// TwinCAT 3 PLC project Plc
// ProgramVersion: 3.1.4024.0
// libraries:
//   Tc2_Standard, * (Beckhoff Automation GmbH)
//   Tc2_System, * (Beckhoff Automation GmbH)
//   Tc3_Module, * (Beckhoff Automation GmbH)
//   VisuSymbols,3.5.10.0,System
// project tree:
//   DUTs/ E_States.TcDUT
//   / Gestore di visualizzazione.TcVMO (not stored), GlobalTextList.TcGTLO, PlcTask.TcTTO
//   GVLs/ Gvl.TcGVL
//   POUs/ FB_StateMachine.TcPOU, MAIN.TcPOU
//   VISUs/ Visualization.TcVIS
// real-time tasks:
//   TASK PlcTask: cycle T#10ms, priority 20, ADS port 350

CONFIGURATION Plc
    RESOURCE PLC ON TwinCAT3
        TASK PlcTask(INTERVAL := T#10ms, PRIORITY := 20);
        PROGRAM MAIN WITH PlcTask : MAIN;
    END_RESOURCE
END_CONFIGURATION

// ---- DUTs/E_States.TcDUT
{attribute 'qualified_only'}
{attribute 'strict'}
TYPE E_States :
(
	eStop := 0,
	eGreen,
	eYellow,
	eRed
);
END_TYPE

// ---- GVLs/Gvl.TcGVL
{attribute 'qualified_only'}
VAR_GLOBAL
	bStart: BOOL; //Pulsante di Start
	bStop: BOOL; //Pulsante di Stop
	Green: BOOL; //Spia verde
	Yellow: BOOL; //Spia verde
	Red: BOOL; //Spia verde
END_VAR

// ---- POUs/MAIN.TcPOU
PROGRAM MAIN
VAR
	StateMachine: FB_StateMachine;
END_VAR

StateMachine(bStart:= Gvl.bStart, bStop:= Gvl.bStop);
//Scrivo gli output
Gvl.Green := StateMachine.Green;
Gvl.Yellow := StateMachine.Yellow;
Gvl.Red := StateMachine.Red;

END_PROGRAM

// ---- POUs/FB_StateMachine.TcPOU
FUNCTION_BLOCK FB_StateMachine
VAR_INPUT
	bStart: BOOL;
	bStop: BOOL;
END_VAR
VAR_OUTPUT
	Green: BOOL;
	Yellow: BOOL;
	Red: BOOL;
END_VAR
VAR
	State: E_States;
	T_Green: TON;
	T_Yellow: TON;
	T_Red: TON;
END_VAR

IF (bStop) THEN
	State:= E_States.eStop;
	//Reset dei timer
	T_Green(IN:= FALSE);
	T_Yellow(IN:= FALSE);
	T_Red(IN:= FALSE);
END_IF

CASE State OF
	E_States.eStop:
		Green:= FALSE;
		Yellow:= FALSE;
		Red:= FALSE;
		IF (NOT bStop AND bSTart) THEN
			State := E_States.eGreen; //Passo allo stato Verde
		END_IF
	
	E_States.eGreen:
		T_Green(IN:= TRUE, PT:= T#5S);
		Green:= TRUE;
		Yellow:= FALSE;
		Red:= FALSE;
		IF (T_Green.Q) THEN //Il tempo del verde è scaduto
			T_Green(IN:= FALSE); //Reset del timer verde 
			State := E_States.eYellow; //Passo allo stato Giallo
		END_IF

	E_States.eYellow:
		T_Yellow(IN:= TRUE, PT:= T#2S);
		Green:= TRUE;
		Yellow:= TRUE;
		Red:= FALSE;
		IF (T_Yellow.Q) THEN //Il tempo del giallo è scaduto
			T_Yellow(IN:= FALSE); //Reset del timer giallo 
			State := E_States.eRed; //Passo allo stato Rosso
		END_IF
		
	E_States.eRed:
		T_Red(IN:= TRUE, PT:= T#8S);
		Green:= FALSE;
		Yellow:= FALSE;
		Red:= TRUE;
		IF (T_Red.Q) THEN //Il tempo del rosso è scaduto
			T_Red(IN:= FALSE); //Reset del timer rosso 
			State := E_States.eGreen; //Passo allo stato Verde
		END_IF
	
END_CASE

END_FUNCTION_BLOCK

// ---- GlobalTextList.TcGTLO
TEXTLIST GlobalTextList
  615 = 'START'
  519 = 'STOP'
END_TEXTLIST

// ---- VISUs/Visualization.TcVIS
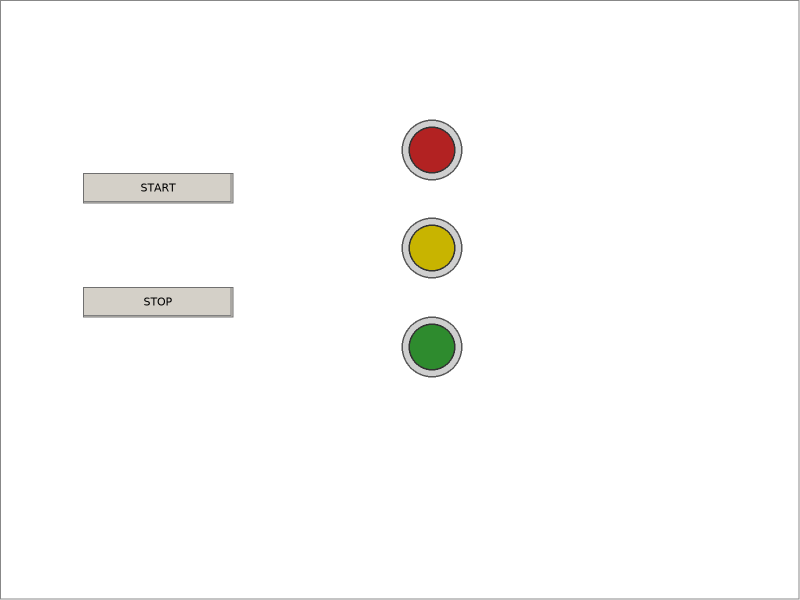
VISUALIZATION Visualization  // 800x600
    Button (83,173 150x30), "START"
        tap Gvl.bStart
    Button (83,287 150x30), "STOP"
        tap Gvl.bStop
    Lamp1 (397,213 70x70), variable: Gvl.Yellow, style: Lamp-Lamp1-Yellow
    Lamp1 (397,115 70x70), variable: Gvl.Red, style: Lamp-Lamp1-Red
    Lamp1 (397,312 70x70), variable: Gvl.Green, style: Lamp-Lamp1-Green
END_VISUALIZATION
